// Block: Area0301_V_Counter

DATA_BLOCK Area0301_V_Counter
VERSION : 0.1
   NON_RETAIN
   VAR
      Value : LReal;
   END_VAR

BEGIN
   // No initialization required
END_DATA_BLOCK
